{attribute 'qualified_only'}
VAR_GLOBAL
	TcJoy : FB_TcJoy;
END_VAR

(* stored: Version 1.1.0.1, ProductVersion 3.1.4019.2
   GVL Global_Variables: Id {3d4ea763-d46a-4a6c-8c86-663c0c89768b} *)
